SYSTEM Projeto_499
  (* Version 1.0, 2024-12-17, Bruno *)
  APPLICATION Projeto_499App
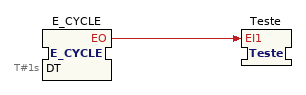
    FBS
      Teste : Teste;
      E_CYCLE : E_CYCLE(DT := T#1s);
    END_FBS
    EVENT_CONNECTIONS
      E_CYCLE.EO TO Teste.EI1;
    END_CONNECTIONS
  END_APPLICATION
  DEVICE FORTE_PC : FORTE_PC(MGR_ID := "localhost:61499")
    {SET_ATTRIBUTE(Profile, HOLOBLOC)} (* device profile *)
    RESOURCE EMB_RES : EMB_RES
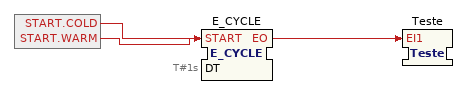
      FBS
        E_CYCLE : E_CYCLE(DT := T#1s);
        Teste : Teste;
      END_FBS
      EVENT_CONNECTIONS
        E_CYCLE.EO TO Teste.EI1;
        START.COLD TO E_CYCLE.START;
        START.WARM TO E_CYCLE.START;
      END_CONNECTIONS
    END_RESOURCE
  END_DEVICE
  MAPPINGS
    Projeto_499App.E_CYCLE ON FORTE_PC.EMB_RES.E_CYCLE;
    Projeto_499App.Teste ON FORTE_PC.EMB_RES.Teste;
  END_MAPPINGS
  SEGMENTS
    Ethernet : Ethernet;
  END_SEGMENTS
  LINKS
    FORTE_PC => Ethernet;
  END_LINKS
END_SYSTEM
